PROGRAM main
  VAR
    STOP : BOOL := 0;
    START : BOOL := 1;
    MOTOR : BOOL;
  END_VAR

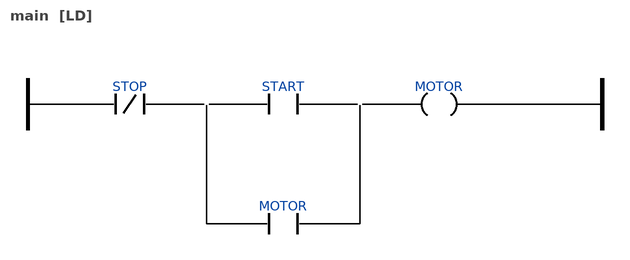
(* LD diagram, written out as Structured Text *)
MOTOR := NOT STOP AND (START OR MOTOR);
END_PROGRAM
